// TwinCAT 3 PLC project EtherCatDiagnosticsSample
// ProgramVersion: 3.1.4026.24
// CompilerDefines: VISU_USEPROPERTYINFO
// libraries:
//   SPT Base Types, * (Beckhoff Automation LLC)
//   SPT EtherCat, * (Beckhoff Automation LLC)
//   SPT Event Logger, * (Beckhoff Automation LLC)
//   Tc2_EtherCAT, * (Beckhoff Automation GmbH)
//   Tc2_Standard, * (Beckhoff Automation GmbH)
//   Tc2_System, * (Beckhoff Automation GmbH)
//   Tc3_EventLogger, * (Beckhoff Automation GmbH)
//   Tc3_PackML_V3, * (Beckhoff Automation GmbH)
// project tree:
//   / GlobalTextList.TcGTLO, PlcTask.TcTTO, Visualization Manager.TcVMO (not stored), Visualization.TcVIS
//   POUs/ MAIN.TcPOU
//   POUs/Modules/00 Machine/ Machine.TcPOU
// real-time tasks:
//   TASK PlcTask: cycle T#10ms, priority 20, ADS port 350
// I/O:
//   DEVICE Device 1 (EtherCAT), AmsNetId 192.168.8.100.5.1
//     Term 1 (EK1100) [EK1100 EtherCAT Coupler (2A E-Bus)]
//       Term 2 (EL6910) [EL6910, TwinSAFE PLC]
//       Term 9 (EL9011) [EL9011 End Terminal]
// variable links:
//   (this object) <-> Device 1 (EtherCAT)
//     PlcTask Inputs/MAIN.MachineModule.MainMaster.EtherCatMaster.AmsNetID <-> InfoData/AmsNetId
//     PlcTask Inputs/MAIN.MachineModule.MainMaster.EtherCatMaster.CfgSlaveCount <-> InfoData/CfgSlaveCount
//     PlcTask Inputs/MAIN.MachineModule.MainMaster.EtherCatMaster.ChangeCount <-> InfoData/ChangeCount
//     PlcTask Inputs/MAIN.MachineModule.MainMaster.EtherCatMaster.DevID <-> InfoData/DevId
//     PlcTask Inputs/MAIN.MachineModule.MainMaster.EtherCatMaster.DevState <-> Inputs/DevState
//     PlcTask Inputs/MAIN.MachineModule.MainMaster.EtherCatMaster.SlaveCount <-> Inputs/SlaveCount
//     PlcTask Inputs/MAIN.MachineModule.MainMaster.FrmXWcState[0] <-> Inputs/Frm0WcState
//     PlcTask Inputs/MAIN.MachineModule.MainSyncUnit.SyncUnitTaskInfo.ObjectId <-> SyncUnits/<default>/<unreferenced>/InfoData/ObjectId
//     PlcTask Inputs/MAIN.MachineModule.MainSyncUnit.SyncUnitTaskInfo.SlaveCount <-> SyncUnits/<default>/<unreferenced>/InfoData/SlaveCount
//     PlcTask Inputs/MAIN.MachineModule.MainSyncUnit.SyncUnitTaskInfo.State <-> SyncUnits/<default>/<unreferenced>/InfoData/State
//     PlcTask Inputs/MAIN.MachineModule.MainSyncUnit.SyncUnitTaskInfo.WcState <-> SyncUnits/<default>/<unreferenced>/WcState/WcState

CONFIGURATION EtherCatDiagnosticsSample
    RESOURCE PLC ON TwinCAT3
        TASK PlcTask(INTERVAL := T#10ms, PRIORITY := 20);
        PROGRAM MAIN WITH PlcTask : MAIN;
    END_RESOURCE
END_CONFIGURATION

// ---- POUs/MAIN.TcPOU
PROGRAM MAIN
VAR
	MachineModule : Machine := (Name := 'Machine');
END_VAR

MachineModule.CyclicLogic();

END_PROGRAM

// ---- POUs/Modules/00 Machine/Machine.TcPOU
FUNCTION_BLOCK Machine EXTENDS FB_PackML_BaseModule
VAR
	// Link EtherCatMaster.* and FrmXWcState[] to the master - see Documentation
	MainMaster : FB_Component_EtherCatMaster := (Name := 'EtherCAT Main');

	// Link SyncUnitTaskInfo.* to the sync unit. Registers itself with MainMaster, which calls it
	MainSyncUnit : FB_SyncUnitTask(EtherCatMaster := MainMaster);
END_VAR

(*
    Machine module. MainMaster is a registered component: its events set
    CurrentAlarmSeverity, and ParentResponseDefinitions decides the PackML reaction.
*)

(* Automatically enables and disables HMI control based on the PackML mode*)
METHOD PROTECTED HMIPermissions
AllowHMIControl(TRUE);
END_METHOD

METHOD PROTECTED Initialize : BOOL
VAR
	Responses : ARRAY[0..4] OF E_AlarmResponse;
END_VAR
Initialize := FALSE;

CASE DescendantSequenceState OF
	0:
		// Framework defaults, stated here so there is one obvious place to change the reaction
		Responses[TcEventSeverity.Verbose]  := E_AlarmResponse.NoResponse;
		Responses[TcEventSeverity.Info]     := E_AlarmResponse.NoResponse;
		Responses[TcEventSeverity.Warning]  := E_AlarmResponse.NoResponse;
		Responses[TcEventSeverity.Error]    := E_AlarmResponse.Abort_ImmediateError;
		Responses[TcEventSeverity.Critical] := E_AlarmResponse.Abort_ImmediateError;
		MainMaster.ParentResponseDefinitions := Responses;

		RegisterComponent(Component := MainMaster);
		DescendantSequenceState := DescendantSequenceState + 10;

	10:
		IF SUPER^.Initialize() THEN
			Initialize := TRUE;
		END_IF
END_CASE
END_METHOD

END_FUNCTION_BLOCK

// ---- Visualization.TcVIS
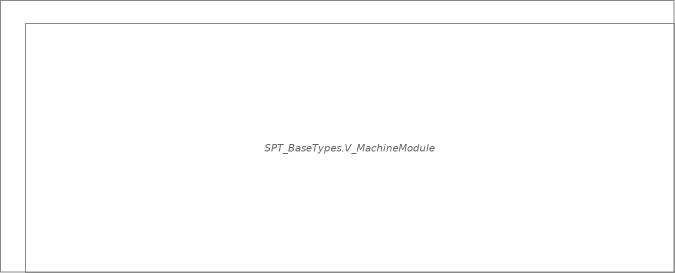
VISUALIZATION Visualization  // 675x273
    Frame (25,23 650x250)
        shows SPT_BaseTypes.V_MachineModule(HMI := MAIN.MachineModule.PackMLBaseModule_HMI)
END_VISUALIZATION
